// TIA Portal V20 export
TYPE "typeSequenceControlNodeJobInterface"
// stored: Namespace Unit1.Em1
   STRUCT
      commands { ExternalWritable := 'False'} : "Unit1.Em1.typeSequenceControlNodeJobInterfaceCommands";
      monitoring { ExternalWritable := 'False'} : "Unit1.Em1.typeSequenceControlNodeJobInterfaceMonitoring";
   END_STRUCT;
END_TYPE
